// TwinCAT 3 PLC project DemoTwinCAT
// ProgramVersion: 3.1.4026.18
// libraries:
//   Tc2_Standard, * (Beckhoff Automation GmbH)
//   Tc2_System, * (Beckhoff Automation GmbH)
// project tree:
//   / PlcTask.TcTTO
//   POUs/ MAIN.TcPOU
// real-time tasks:
//   TASK PlcTask: cycle T#10ms, priority 20, ADS port 350

CONFIGURATION DemoTwinCAT
    RESOURCE PLC ON TwinCAT3
        TASK PlcTask(INTERVAL := T#10ms, PRIORITY := 20);
        PROGRAM MAIN WITH PlcTask : MAIN;
    END_RESOURCE
END_CONFIGURATION

// ---- POUs/MAIN.TcPOU
PROGRAM MAIN
VAR
    // Simpele demo: twee schakelaars en een lampje
    // Zet in online mode bSwitch1/bSwitch2 aan/uit en kijk hoe bLamp reageert

    bSwitch1       : BOOL := FALSE;   // Schakelaar 1 (input)
    bSwitch2       : BOOL := FALSE;   // Schakelaar 2 (input)
    bEmergencyStop : BOOL := FALSE;   // Noodstop – forceert lamp uit
    bLamp          : BOOL := FALSE;   // Lamp (output)	
	Implementation: BOOL;
	POU: BOOL;
	TcPlcObject: BOOL;
END_VAR

// =============================================
// MAIN - Simpele demo met schakelaars en lampje TEST
// =============================================

// Logica: lamp aan als een van de schakelaars waar is,
// tenzij de noodstop actief is (dan altijd uit)
IF bEmergencyStop THEN
    bLamp := FALSE;
ELSE
    bLamp := bSwitch1 OR bSwitch2;
END_IF;

END_PROGRAM
